(* Schneider Machine Expert - Basic project Modelo final v1.2, file version 2.5.0.0 *)
(* ProjectInformations: Name=Nuevo proyecto *)

HARDWARE
  Cpu 0: TM221CE24T
  EthernetConfiguration: NetworkName=M221, IpAllocationMode=FixedAddress, IpAddress=0.0.0.0, SubnetMask=0.0.0.0
  SerialLineConfiguration: Baud=Baud19200, Parity=ParityEven, DataBits=DataBits8, StopBits=StopBits1, PhysicalMedium=PhysicalMediumRs485, TransmissionMode=TransmissionModeModbusRtu, SlaveId=1, Addressing=SlaveAddressing
  MastTask: UsePeriodScanMode=false, PeriodScan=100
  FastTask: Period=255
  CpuBehavior: StartingMode=StartAsPreviousState, AutoSaveRamOnEeprom=true, WatchdogPeriod=250

SYMBOLS  (address, symbol, comment, settings)
  %M0         "Escalon frontal izquierdo"
  %M1         "Escalon frontal derecho"
  %M2         "Escalon trasero izquierdo"
  %M3         "Escalon trasero derecho"
  %M4         "Sensor frente izquierdo"
  %M5         "Sensor frente medio"
  %M6         "Sensor frente derecho"
  %M7         "Sensor derecha adelante"
  %M8         "Sensor derecha medio"
  %M9         "Sensor derecha atras"
  %M10        "Sensor trasero derecha"
  %M11        "Sensor trasero medio"
  %M12        "Sensor trasero izquierda"
  %M13        "Sensor izquierda atras"
  %M14        "Sensor izquierda medio"
  %M15        "Sensor izquierda adelante"
  %M16      FIFO_IN  "Carga en fifo"
  %M17      FIFO_OUT  "Descarga de fifo"
  %M40      RST_S  "Reset/Enable Generador S"
  %M41      RST_DEMUX  "Reset/Enbale Demux"
  %M42      EN_ENCOD  "Enable Encoders"
  %M43      RST_ENCOD  "Reset Encoders"
  %M44      RST_FIFO  "Reset FIFOS"
  %M45      RST_STOP
  %M50      STP_MOV  "Stop Movement"
  %M51        "Enable Forward"
  %M52        "Enable Giro Horario"
  %M53        "Enable Giro A-Horario"
  %M54        "Enable F-G-H"
  %M55        "Enable F-G-AH"
  %M56        "Enable B-G-H"
  %M57        "Enable B-G-AH"
  %S6       SB_TB1S  "Base de tiempo de 1 s generada por un reloj interno"
  %MW10       "Comando Rueda Izquierda"
  %MW11       "Comando Rueda Derecha"
  %MW12       "Velocidad Rueda Izquierda"
  %MW13       "Velocidad Rueda Derecha"
  %TM0        [Preset=5, Base=OneHundredMilliSeconds]
  %TM1        [Preset=5, Base=OneHundredMilliSeconds]
  %TM2        [Preset=5, Base=OneHundredMilliSeconds]
  %TM3        [Preset=5, Base=OneHundredMilliSeconds]
  %TM4        [Preset=5, Base=OneHundredMilliSeconds]
  %TM5        [Preset=5, Base=OneHundredMilliSeconds]
  %TM6        [Preset=5, Base=OneHundredMilliSeconds]
  %TM7        [Preset=5, Base=OneHundredMilliSeconds]
  %TM8        [Preset=5, Base=OneHundredMilliSeconds]
  %TM9        [Preset=5, Base=OneHundredMilliSeconds]
  %TM10       [Preset=5, Base=OneHundredMilliSeconds]
  %TM11       [Preset=5, Base=OneHundredMilliSeconds]
  %TM12       [Preset=5, Base=OneHundredMilliSeconds]
  %TM13       [Preset=5, Base=OneHundredMilliSeconds]
  %TM14       [Preset=5, Base=OneHundredMilliSeconds]
  %TM15       [Preset=5, Base=OneHundredMilliSeconds]
  %C0         [Preset=17]
  %R0         "Pasos Izquierda"
  %R1         "Pasos Derecha"
  %R2         "Velocidad Izquierda"
  %R3         "Velocidad Derecha"
  %UDF0.RETF0   "Orientacion"  [CompiledType=Float, Type=ReturnValue, DisplayedAddress=%RET0, CompiledAddress=%UDFRETURNF0]
  %UDF0.VARF0   "Cuenta encoder L"  [CompiledType=Float, Type=Variable, DisplayedAddress=%VAR0, CompiledAddress=%UDFVARF0]
  %UDF0.VARF1   "Cuenta Encoder R"  [CompiledType=Float, Type=Variable, DisplayedAddress=%VAR1, CompiledAddress=%UDFVARF1]
  %UDF0.VARF2   "Radio de la Rueda"  [CompiledType=Float, Type=Variable, DisplayedAddress=%VAR2, CompiledAddress=%UDFVARF2]
  %UDF0.VARF4   "Pasos"  [CompiledType=Float, Type=Variable, DisplayedAddress=%VAR4, CompiledAddress=%UDFVARF4]
  %UDF0.VARF6   "ΔSL"  [CompiledType=Float, Type=Variable, DisplayedAddress=%VAR6, CompiledAddress=%UDFVARF6]
  %UDF0.VARF7   "ΔSR:"  [CompiledType=Float, Type=Variable, DisplayedAddress=%VAR7, CompiledAddress=%UDFVARF7]
  %UDF0.VARF9   "Longitud Eje"  [CompiledType=Float, Type=Variable, DisplayedAddress=%VAR9, CompiledAddress=%UDFVARF9]
  %I0.0     ENC1A  "Input"
  %I0.1     ENC1B  "Enable"
  %I0.6     ENC2A
  %I0.7     ENC2B
  %I0.8     MUX_IN  "Data de mux sensores"
  %Q0.0     L_PWM  "Salida PWM Motor Izquierdo"
  %Q0.1     R_PWM  "Salida PWM Motor Derecho"
  %Q0.2     L_DIR  "Salida Direccion Motor Izquierdo - 0:F 1:B"
  %Q0.3     R_DIR  "Salida Direccion Motor Derecho - 0:F 1:B"
  %Q0.4     S0  "MUX S0"
  %Q0.5     S1  "MUX S1"
  %Q0.6     S2  "MUX S2"
  %Q0.7     S3  "MUX S3"
  %Q0.8       "LAMPARAS BIT 0"
  %Q0.9       "LAMPARAS BIT 1"
  %HSC0       "Encoder Rueda Izquierda"  [Type=CounterOrDownCounterBiPhasesX2, Preset=0, UseDoubleWord=true, DedicatedInputs(DedicatedInput(Activated=true), DedicatedInput(Activated=true)), ReflexOutputs(ReflexOutput(Activated=false, LessThanS0=false, GreaterOrEqualThanS0=false, GreaterOrEqualThanS1=false), ReflexOutput(Activated=false, LessThanS0=false, GreaterOrEqualThanS0=false, GreaterOrEqualThanS1=false)), Thresholds(Threshold(Thresh]
  %HSC1       "Encoder Rueda Derecha"  [Type=CounterOrDownCounterBiPhasesX2, Preset=0, UseDoubleWord=true, DedicatedInputs(DedicatedInput(Activated=true), DedicatedInput(Activated=true)), ReflexOutputs(ReflexOutput(Activated=false, LessThanS0=false, GreaterOrEqualThanS0=false, GreaterOrEqualThanS1=false), ReflexOutput(Activated=false, LessThanS0=false, GreaterOrEqualThanS0=false, GreaterOrEqualThanS1=false)), Thresholds(Threshold(Thresh]
  %PWM0       "PWM_L"  [PtoObject(RefInput=NotUsed, ZPhaseInput=NotUsed, ProbeInput=NotUsed), GlobalIndex=0, Type=PWM, TimeBase=OneMilliSeconds, Preset=1]
  %PWM1       "PWM_R"  [PtoObject(RefInput=NotUsed, ZPhaseInput=NotUsed, ProbeInput=NotUsed), GlobalIndex=1, Type=PWM, TimeBase=OneMilliSeconds, Preset=1]

POU Demux
  (* SectionNumber=1 *)

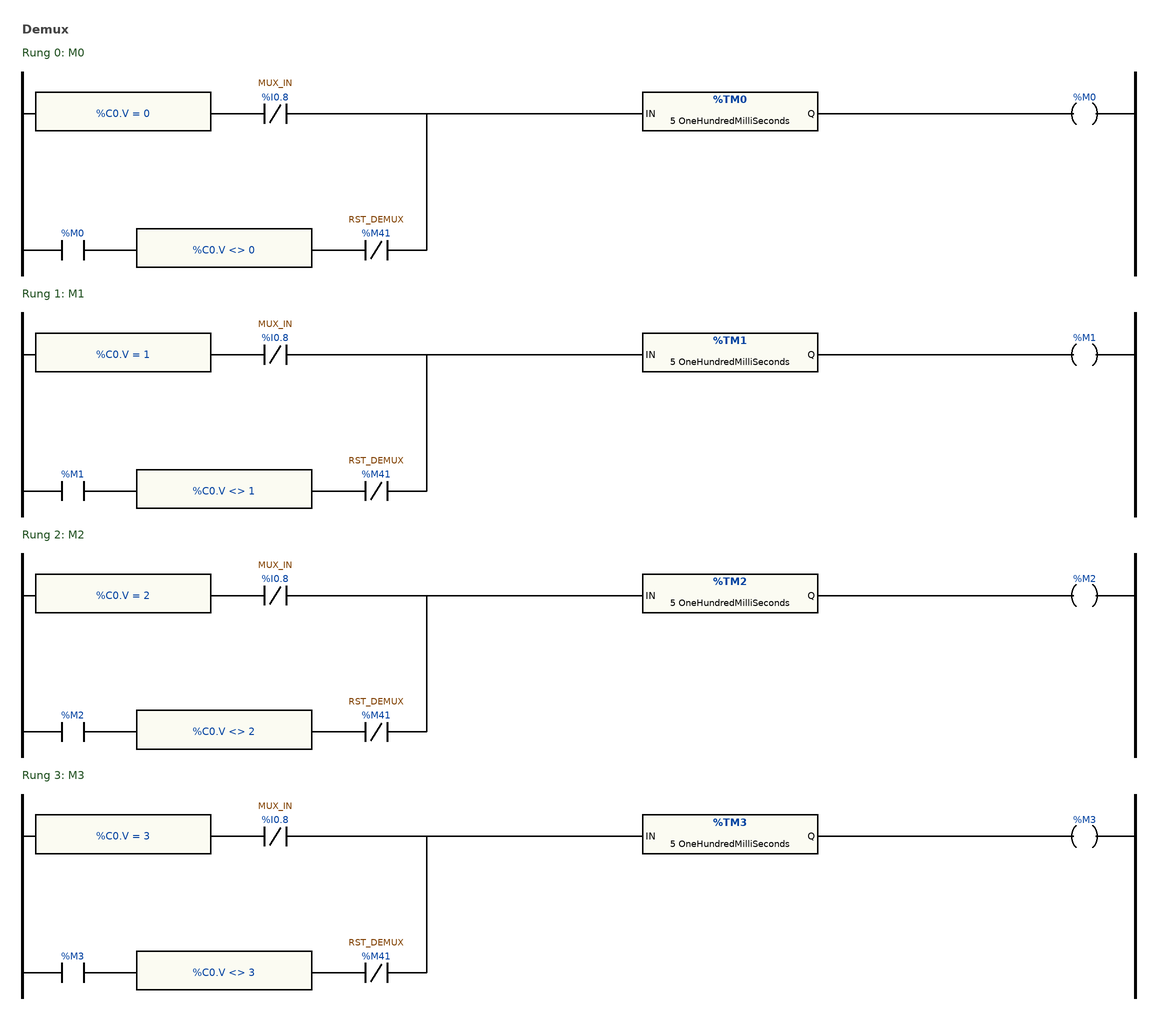

// Rung 0: M0
  BLK %TM0
  LD [ %C0.V = 0 ]
  ANDN %I0.8              (* MUX_IN *)
  OR( %M0
  AND [ %C0.V <> 0 ]
  ANDN %M41               (* RST_DEMUX *)
  )
  IN
  OUT_BLK
  LD Q
  ST %M0
  END_BLK
  // as ST:
  //   %TM0(IN := %C0.V = 0 AND NOT MUX_IN OR %M0 AND %C0.V <> 0 AND NOT RST_DEMUX);
  //   %M0 := %TM0.Q;

// Rung 1: M1
  BLK %TM1
  LD [ %C0.V = 1 ]
  ANDN %I0.8              (* MUX_IN *)
  OR( %M1
  AND [ %C0.V <> 1 ]
  ANDN %M41               (* RST_DEMUX *)
  )
  IN
  OUT_BLK
  LD Q
  ST %M1
  END_BLK
  // as ST:
  //   %TM1(IN := %C0.V = 1 AND NOT MUX_IN OR %M1 AND %C0.V <> 1 AND NOT RST_DEMUX);
  //   %M1 := %TM1.Q;

// Rung 2: M2
  BLK %TM2
  LD [ %C0.V = 2 ]
  ANDN %I0.8              (* MUX_IN *)
  OR( %M2
  AND [ %C0.V <> 2 ]
  ANDN %M41               (* RST_DEMUX *)
  )
  IN
  OUT_BLK
  LD Q
  ST %M2
  END_BLK
  // as ST:
  //   %TM2(IN := %C0.V = 2 AND NOT MUX_IN OR %M2 AND %C0.V <> 2 AND NOT RST_DEMUX);
  //   %M2 := %TM2.Q;

// Rung 3: M3
  BLK %TM3
  LD [ %C0.V = 3 ]
  ANDN %I0.8              (* MUX_IN *)
  OR( %M3
  AND [ %C0.V <> 3 ]
  ANDN %M41               (* RST_DEMUX *)
  )
  IN
  OUT_BLK
  LD Q
  ST %M3
  END_BLK
  // as ST:
  //   %TM3(IN := %C0.V = 3 AND NOT MUX_IN OR %M3 AND %C0.V <> 3 AND NOT RST_DEMUX);
  //   %M3 := %TM3.Q;

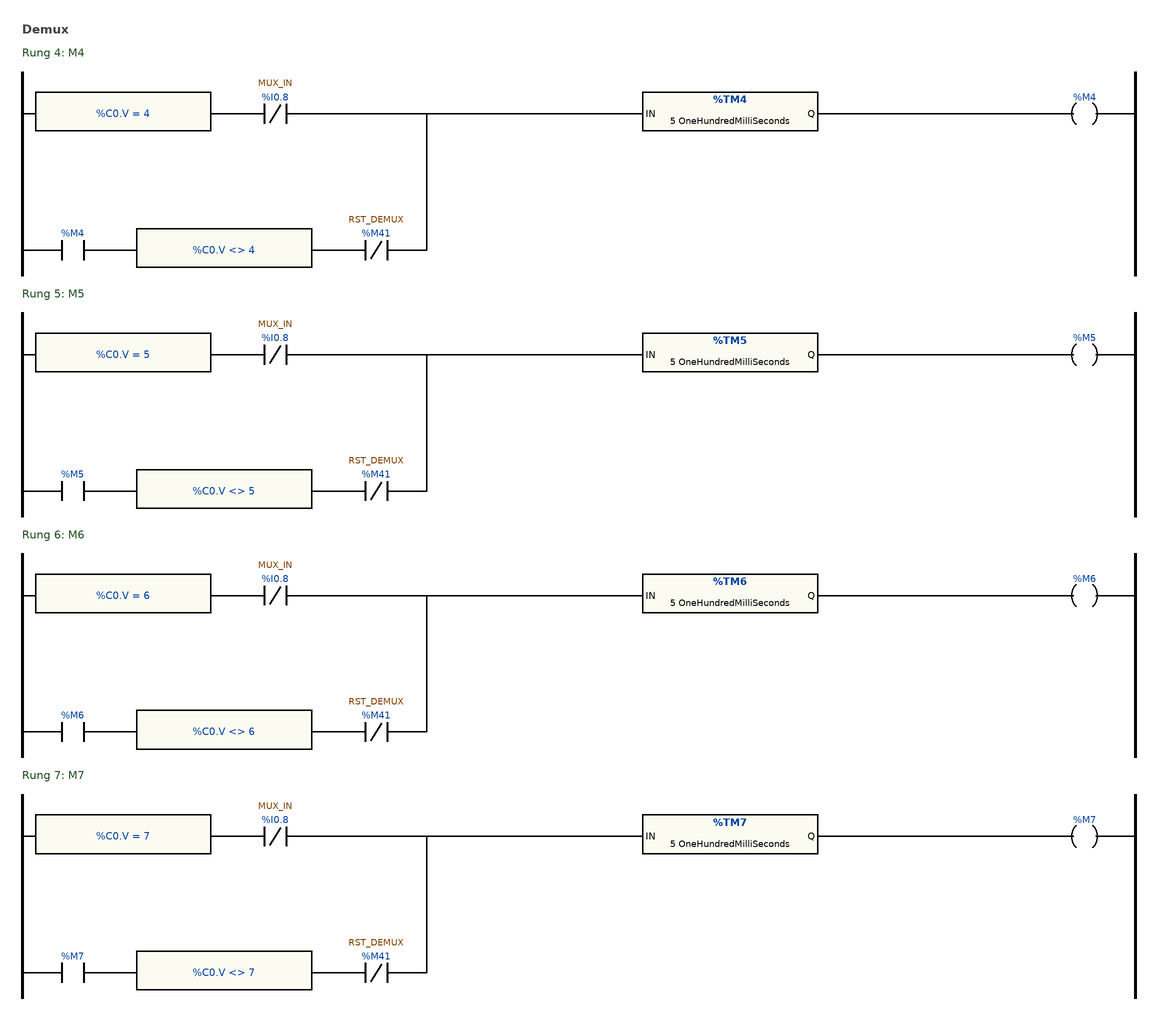

// Rung 4: M4
  BLK %TM4
  LD [ %C0.V = 4 ]
  ANDN %I0.8              (* MUX_IN *)
  OR( %M4
  AND [ %C0.V <> 4 ]
  ANDN %M41               (* RST_DEMUX *)
  )
  IN
  OUT_BLK
  LD Q
  ST %M4
  END_BLK
  // as ST:
  //   %TM4(IN := %C0.V = 4 AND NOT MUX_IN OR %M4 AND %C0.V <> 4 AND NOT RST_DEMUX);
  //   %M4 := %TM4.Q;

// Rung 5: M5
  BLK %TM5
  LD [ %C0.V = 5 ]
  ANDN %I0.8              (* MUX_IN *)
  OR( %M5
  AND [ %C0.V <> 5 ]
  ANDN %M41               (* RST_DEMUX *)
  )
  IN
  OUT_BLK
  LD Q
  ST %M5
  END_BLK
  // as ST:
  //   %TM5(IN := %C0.V = 5 AND NOT MUX_IN OR %M5 AND %C0.V <> 5 AND NOT RST_DEMUX);
  //   %M5 := %TM5.Q;

// Rung 6: M6
  BLK %TM6
  LD [ %C0.V = 6 ]
  ANDN %I0.8              (* MUX_IN *)
  OR( %M6
  AND [ %C0.V <> 6 ]
  ANDN %M41               (* RST_DEMUX *)
  )
  IN
  OUT_BLK
  LD Q
  ST %M6
  END_BLK
  // as ST:
  //   %TM6(IN := %C0.V = 6 AND NOT MUX_IN OR %M6 AND %C0.V <> 6 AND NOT RST_DEMUX);
  //   %M6 := %TM6.Q;

// Rung 7: M7
  BLK %TM7
  LD [ %C0.V = 7 ]
  ANDN %I0.8              (* MUX_IN *)
  OR( %M7
  AND [ %C0.V <> 7 ]
  ANDN %M41               (* RST_DEMUX *)
  )
  IN
  OUT_BLK
  LD Q
  ST %M7
  END_BLK
  // as ST:
  //   %TM7(IN := %C0.V = 7 AND NOT MUX_IN OR %M7 AND %C0.V <> 7 AND NOT RST_DEMUX);
  //   %M7 := %TM7.Q;

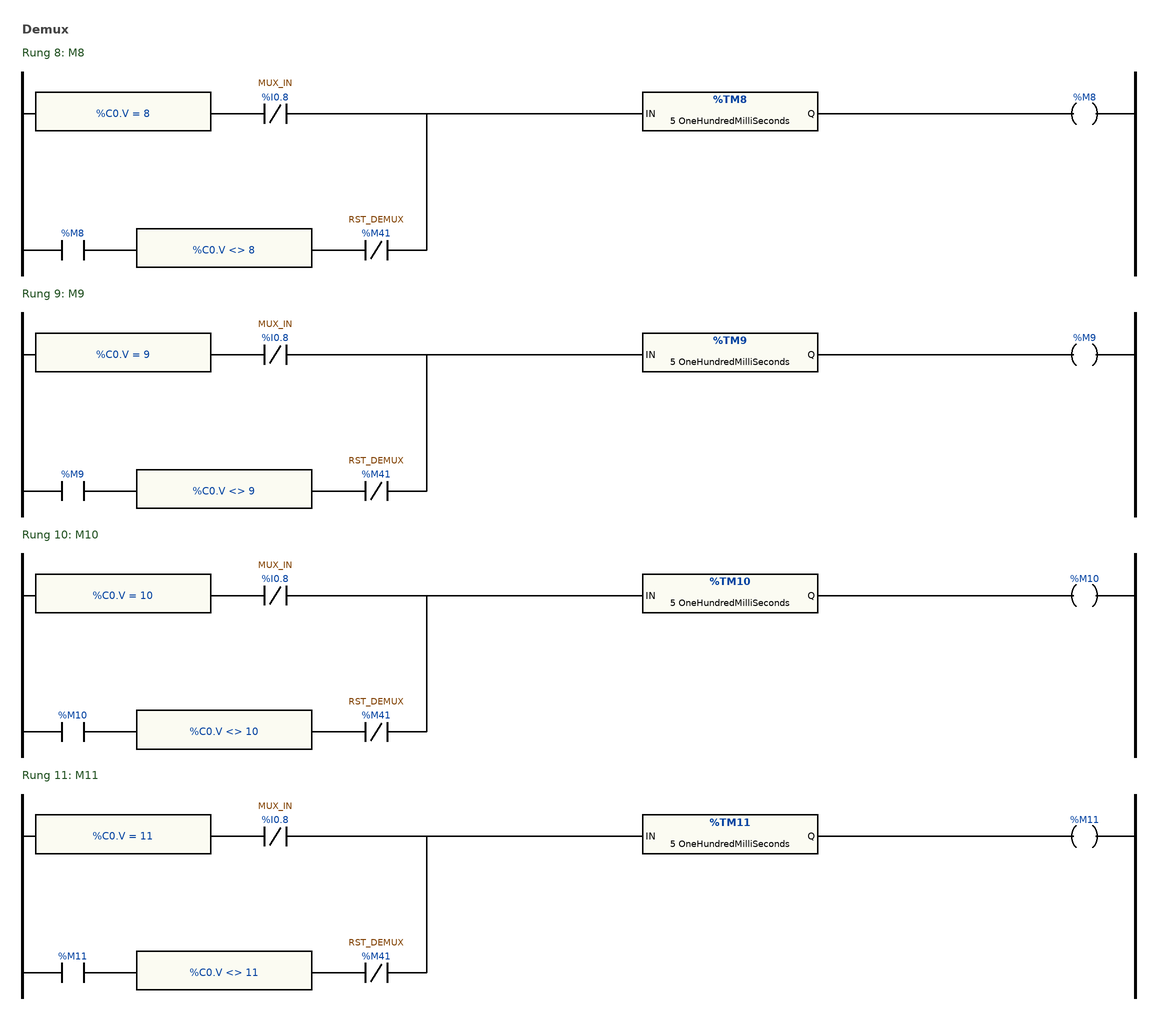

// Rung 8: M8
  BLK %TM8
  LD [ %C0.V = 8 ]
  ANDN %I0.8              (* MUX_IN *)
  OR( %M8
  AND [ %C0.V <> 8 ]
  ANDN %M41               (* RST_DEMUX *)
  )
  IN
  OUT_BLK
  LD Q
  ST %M8
  END_BLK
  // as ST:
  //   %TM8(IN := %C0.V = 8 AND NOT MUX_IN OR %M8 AND %C0.V <> 8 AND NOT RST_DEMUX);
  //   %M8 := %TM8.Q;

// Rung 9: M9
  BLK %TM9
  LD [ %C0.V = 9 ]
  ANDN %I0.8              (* MUX_IN *)
  OR( %M9
  AND [ %C0.V <> 9 ]
  ANDN %M41               (* RST_DEMUX *)
  )
  IN
  OUT_BLK
  LD Q
  ST %M9
  END_BLK
  // as ST:
  //   %TM9(IN := %C0.V = 9 AND NOT MUX_IN OR %M9 AND %C0.V <> 9 AND NOT RST_DEMUX);
  //   %M9 := %TM9.Q;

// Rung 10: M10
  BLK %TM10
  LD [ %C0.V = 10 ]
  ANDN %I0.8              (* MUX_IN *)
  OR( %M10
  AND [ %C0.V <> 10 ]
  ANDN %M41               (* RST_DEMUX *)
  )
  IN
  OUT_BLK
  LD Q
  ST %M10
  END_BLK
  // as ST:
  //   %TM10(IN := %C0.V = 10 AND NOT MUX_IN OR %M10 AND %C0.V <> 10 AND NOT RST_DEMUX);
  //   %M10 := %TM10.Q;

// Rung 11: M11
  BLK %TM11
  LD [ %C0.V = 11 ]
  ANDN %I0.8              (* MUX_IN *)
  OR( %M11
  AND [ %C0.V <> 11 ]
  ANDN %M41               (* RST_DEMUX *)
  )
  IN
  OUT_BLK
  LD Q
  ST %M11
  END_BLK
  // as ST:
  //   %TM11(IN := %C0.V = 11 AND NOT MUX_IN OR %M11 AND %C0.V <> 11 AND NOT RST_DEMUX);
  //   %M11 := %TM11.Q;

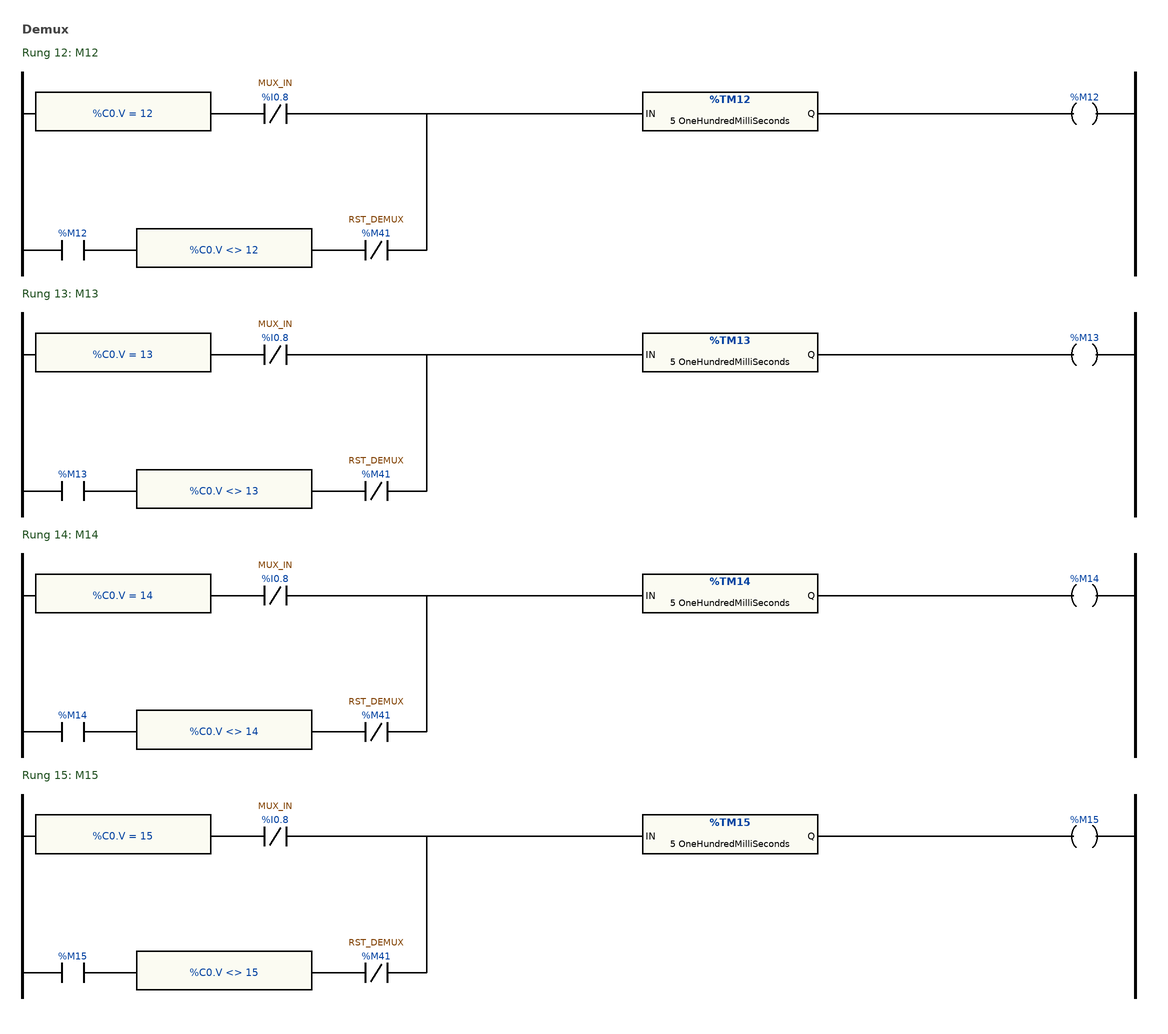

// Rung 12: M12
  BLK %TM12
  LD [ %C0.V = 12 ]
  ANDN %I0.8              (* MUX_IN *)
  OR( %M12
  AND [ %C0.V <> 12 ]
  ANDN %M41               (* RST_DEMUX *)
  )
  IN
  OUT_BLK
  LD Q
  ST %M12
  END_BLK
  // as ST:
  //   %TM12(IN := %C0.V = 12 AND NOT MUX_IN OR %M12 AND %C0.V <> 12 AND NOT RST_DEMUX);
  //   %M12 := %TM12.Q;

// Rung 13: M13
  BLK %TM13
  LD [ %C0.V = 13 ]
  ANDN %I0.8              (* MUX_IN *)
  OR( %M13
  AND [ %C0.V <> 13 ]
  ANDN %M41               (* RST_DEMUX *)
  )
  IN
  OUT_BLK
  LD Q
  ST %M13
  END_BLK
  // as ST:
  //   %TM13(IN := %C0.V = 13 AND NOT MUX_IN OR %M13 AND %C0.V <> 13 AND NOT RST_DEMUX);
  //   %M13 := %TM13.Q;

// Rung 14: M14
  BLK %TM14
  LD [ %C0.V = 14 ]
  ANDN %I0.8              (* MUX_IN *)
  OR( %M14
  AND [ %C0.V <> 14 ]
  ANDN %M41               (* RST_DEMUX *)
  )
  IN
  OUT_BLK
  LD Q
  ST %M14
  END_BLK
  // as ST:
  //   %TM14(IN := %C0.V = 14 AND NOT MUX_IN OR %M14 AND %C0.V <> 14 AND NOT RST_DEMUX);
  //   %M14 := %TM14.Q;

// Rung 15: M15
  BLK %TM15
  LD [ %C0.V = 15 ]
  ANDN %I0.8              (* MUX_IN *)
  OR( %M15
  AND [ %C0.V <> 15 ]
  ANDN %M41               (* RST_DEMUX *)
  )
  IN
  OUT_BLK
  LD Q
  ST %M15
  END_BLK
  // as ST:
  //   %TM15(IN := %C0.V = 15 AND NOT MUX_IN OR %M15 AND %C0.V <> 15 AND NOT RST_DEMUX);
  //   %M15 := %TM15.Q;

POU Generacion Sx
  (* SectionNumber=2 *)

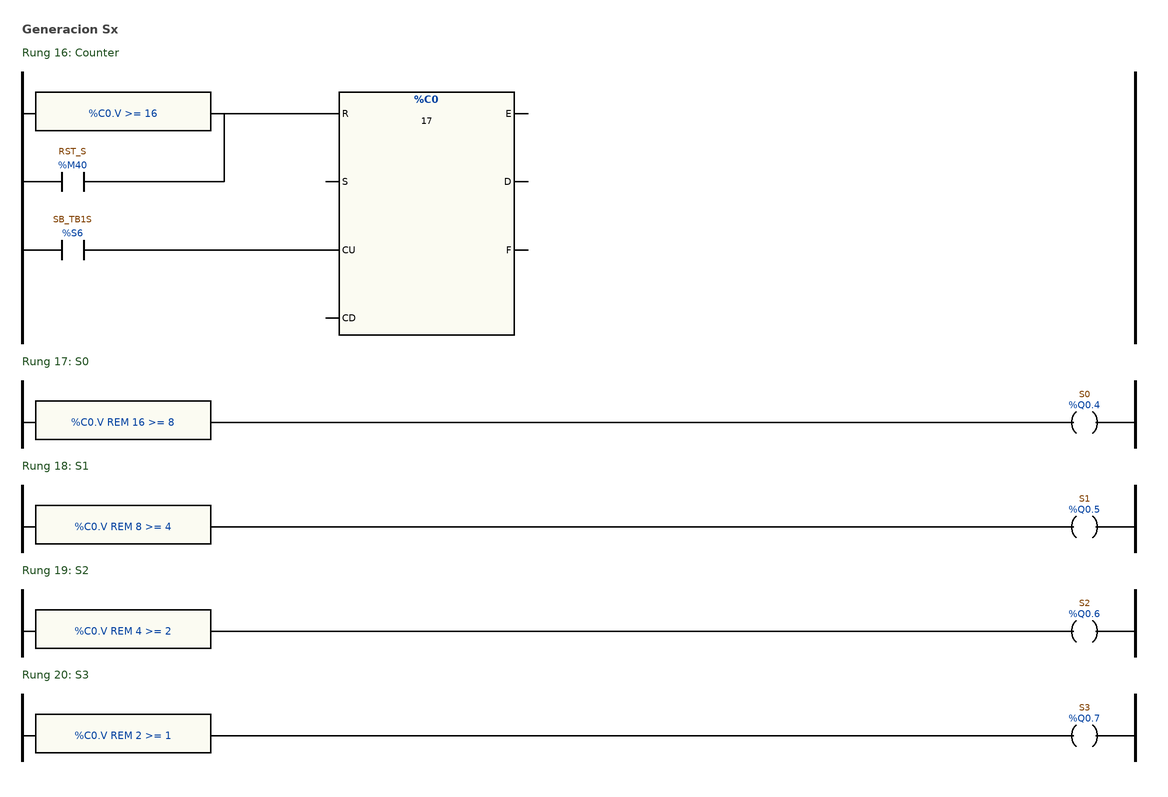

// Rung 16: Counter
  BLK %C0
  LD [ %C0.V >= 16 ]
  OR %M40                 (* RST_S *)
  R
  LD %S6                  (* SB_TB1S *)
  CU
  END_BLK
  // as ST:
  //   %C0(R := %C0.V >= 16 OR RST_S, CU := SB_TB1S);

// Rung 17: S0
  LD 1
  AND [%C0.V REM 16 >= 8]
  ST %Q0.4                (* S0 *)
  // as ST:
  //   S0 := %C0.V REM 16 >= 8;

// Rung 18: S1
  LD 1
  AND [%C0.V REM 8 >= 4]
  ST %Q0.5                (* S1 *)
  // as ST:
  //   S1 := %C0.V REM 8 >= 4;

// Rung 19: S2
  LD 1
  AND [%C0.V REM 4 >= 2]
  ST %Q0.6                (* S2 *)
  // as ST:
  //   S2 := %C0.V REM 4 >= 2;

// Rung 20: S3
  LD 1
  AND [%C0.V REM 2 >= 1]
  ST %Q0.7                (* S3 *)
  // as ST:
  //   S3 := %C0.V REM 2 >= 1;

POU Encoders
  (* SectionNumber=0 *)

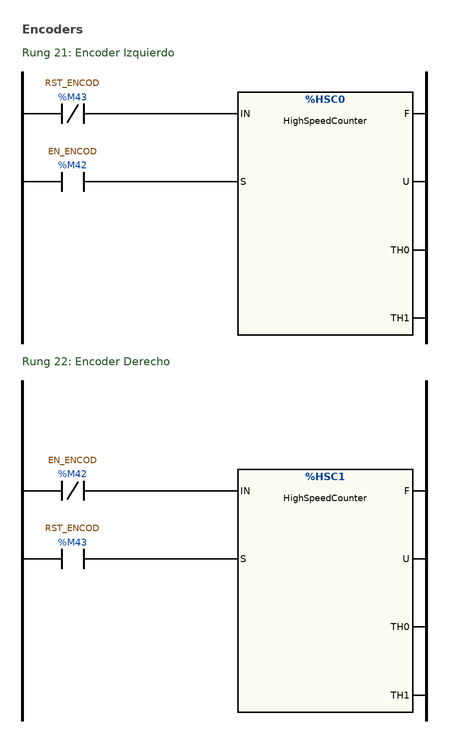

// Rung 21: Encoder Izquierdo
  BLK %HSC0
  LDN %M43                (* RST_ENCOD *)
  IN
  LD %M42                 (* EN_ENCOD *)
  S
  END_BLK
  // as ST:
  //   %HSC0(IN := NOT RST_ENCOD, S := EN_ENCOD);

// Rung 22: Encoder Derecho
  BLK %HSC1
  LDN %M42                (* EN_ENCOD *)
  IN
  LD %M43                 (* RST_ENCOD *)
  S
  END_BLK
  // as ST:
  //   %HSC1(IN := NOT EN_ENCOD, S := RST_ENCOD);

POU Control de Motores
  (* SectionNumber=0 *)

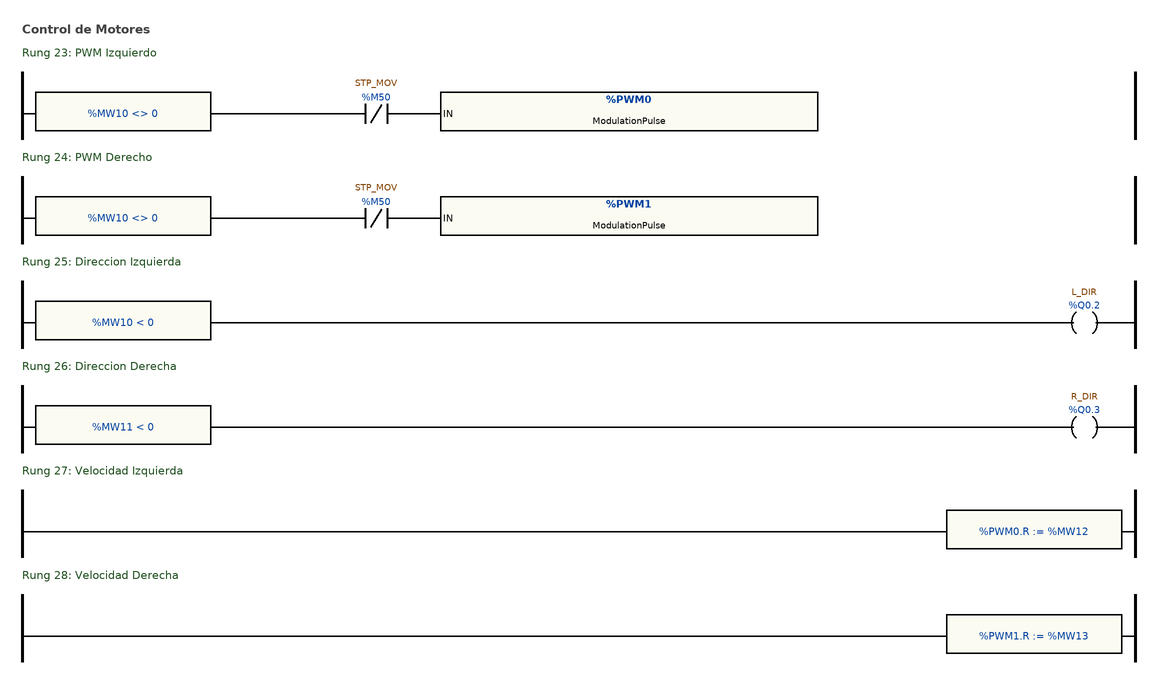

// Rung 23: PWM Izquierdo
  BLK %PWM0
  LD [ %MW10 <> 0 ]
  ANDN %M50               (* STP_MOV *)
  IN
  END_BLK
  // as ST:
  //   %PWM0(IN := %MW10 <> 0 AND NOT STP_MOV);

// Rung 24: PWM Derecho
  BLK %PWM1
  LD [ %MW10 <> 0 ]
  ANDN %M50               (* STP_MOV *)
  IN
  END_BLK
  // as ST:
  //   %PWM1(IN := %MW10 <> 0 AND NOT STP_MOV);

// Rung 25: Direccion Izquierda
  LD [ %MW10 < 0 ]
  ST %Q0.2                (* L_DIR *)
  // as ST:
  //   L_DIR := %MW10 < 0;

// Rung 26: Direccion Derecha
  LD [ %MW11 < 0 ]
  ST %Q0.3                (* R_DIR *)
  // as ST:
  //   R_DIR := %MW11 < 0;

// Rung 27: Velocidad Izquierda
  LD 1
  [ %PWM0.R := %MW12 ]
  // as ST:
  //   %PWM0.R := %MW12;

// Rung 28: Velocidad Derecha
  LD 1
  [ %PWM1.R := %MW13 ]
  // as ST:
  //   %PWM1.R := %MW13;

POU FIFOS
  (* SectionNumber=0 *)

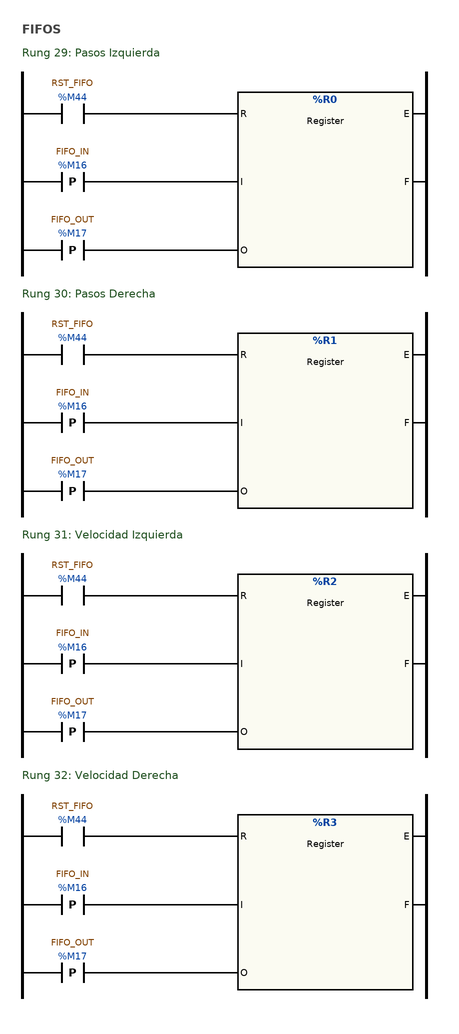

// Rung 29: Pasos Izquierda
  BLK %R0
  LD %M44                 (* RST_FIFO *)
  R
  LDR %M16                (* FIFO_IN *)
  I
  LDR %M17                (* FIFO_OUT *)
  O
  END_BLK
  // as ST:
  //   %R0(R := RST_FIFO, I := RISING(FIFO_IN), O := RISING(FIFO_OUT));

// Rung 30: Pasos Derecha
  BLK %R1
  LD %M44                 (* RST_FIFO *)
  R
  LDR %M16                (* FIFO_IN *)
  I
  LDR %M17                (* FIFO_OUT *)
  O
  END_BLK
  // as ST:
  //   %R1(R := RST_FIFO, I := RISING(FIFO_IN), O := RISING(FIFO_OUT));

// Rung 31: Velocidad Izquierda
  BLK %R2
  LD %M44                 (* RST_FIFO *)
  R
  LDR %M16                (* FIFO_IN *)
  I
  LDR %M17                (* FIFO_OUT *)
  O
  END_BLK
  // as ST:
  //   %R2(R := RST_FIFO, I := RISING(FIFO_IN), O := RISING(FIFO_OUT));

// Rung 32: Velocidad Derecha
  BLK %R3
  LD %M44                 (* RST_FIFO *)
  R
  LDR %M16                (* FIFO_IN *)
  I
  LDR %M17                (* FIFO_OUT *)
  O
  END_BLK
  // as ST:
  //   %R3(R := RST_FIFO, I := RISING(FIFO_IN), O := RISING(FIFO_OUT));

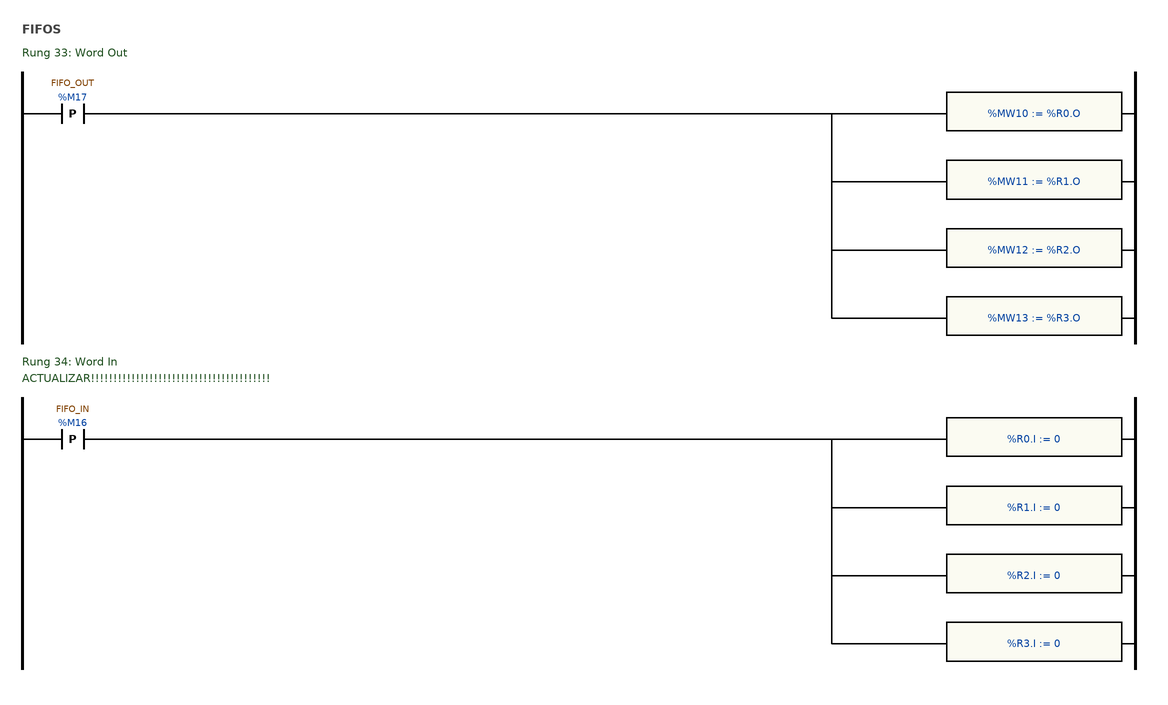

// Rung 33: Word Out
  LDR %M17                (* FIFO_OUT *)
  [ %MW10 := %R0.O ]
  [ %MW11 := %R1.O ]
  [ %MW12 := %R2.O ]
  [ %MW13 := %R3.O ]
  // as ST:
  //   IF RISING(FIFO_OUT) THEN %MW10 := %R0.O; END_IF;
  //   IF RISING(FIFO_OUT) THEN %MW11 := %R1.O; END_IF;
  //   IF RISING(FIFO_OUT) THEN %MW12 := %R2.O; END_IF;
  //   IF RISING(FIFO_OUT) THEN %MW13 := %R3.O; END_IF;

// Rung 34: Word In
// ACTUALIZAR!!!!!!!!!!!!!!!!!!!!!!!!!!!!!!!!!!!!!!!!
  LDR %M16                (* FIFO_IN *)
  [ %R0.I := 0 ]
  [ %R1.I := 0 ]
  [ %R2.I := 0 ]
  [ %R3.I := 0 ]
  // as ST:
  //   IF RISING(FIFO_IN) THEN %R0.I := 0; END_IF;
  //   IF RISING(FIFO_IN) THEN %R1.I := 0; END_IF;
  //   IF RISING(FIFO_IN) THEN %R2.I := 0; END_IF;
  //   IF RISING(FIFO_IN) THEN %R3.I := 0; END_IF;

POU Control de Colision
  (* SectionNumber=0 *)

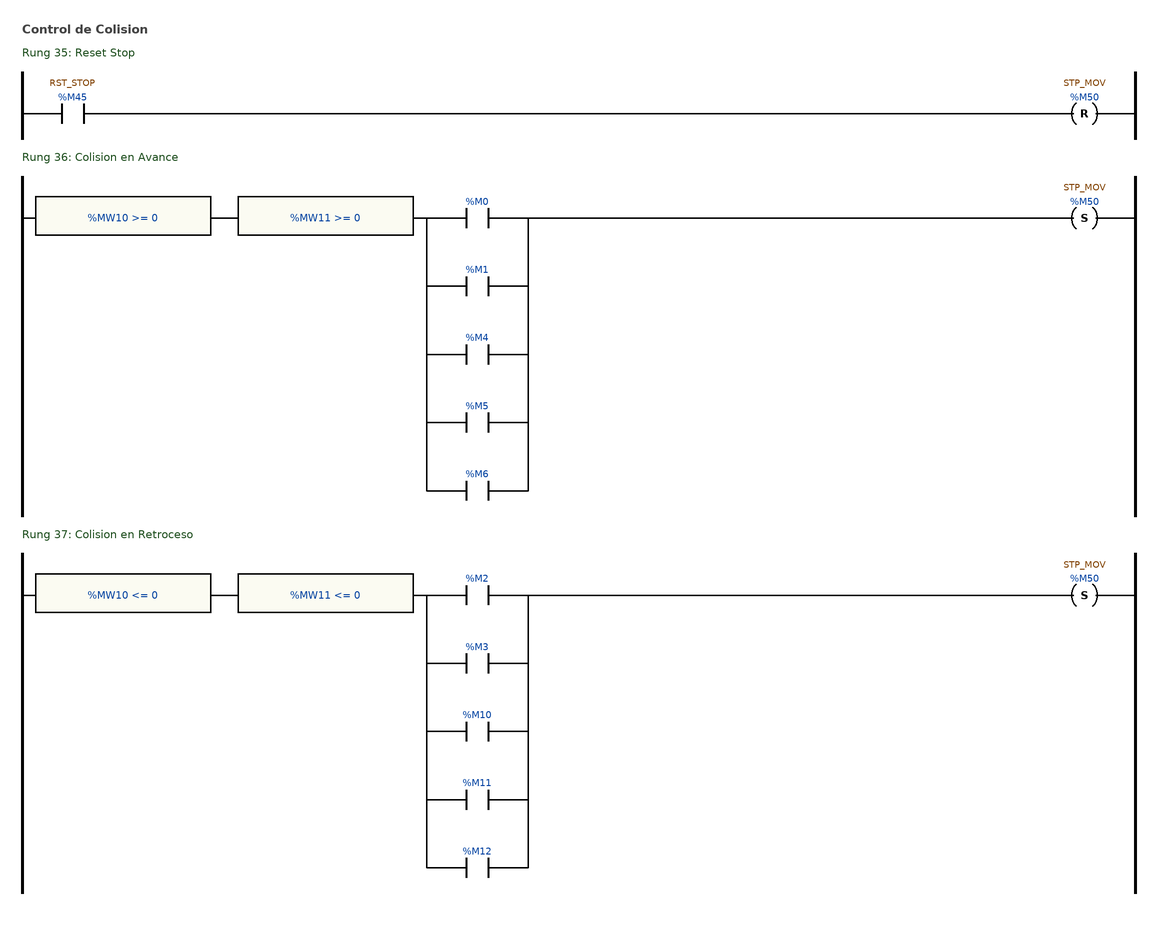

// Rung 35: Reset Stop
  LD %M45                 (* RST_STOP *)
  R %M50                  (* STP_MOV *)
  // as ST:
  //   IF RST_STOP THEN STP_MOV := FALSE; END_IF;

// Rung 36: Colision en Avance
  LD [ %MW10 >= 0 ]
  AND [ %MW11 >= 0 ]
  AND( %M0
  OR %M1
  OR %M4
  OR %M5
  OR %M6
  )
  S %M50                  (* STP_MOV *)
  // as ST:
  //   IF %MW10 >= 0 AND %MW11 >= 0 AND (%M0 OR %M1 OR %M4 OR %M5 OR %M6) THEN STP_MOV := TRUE; END_IF;

// Rung 37: Colision en Retroceso
  LD [ %MW10 <= 0 ]
  AND [ %MW11 <= 0 ]
  AND( %M2
  OR %M3
  OR %M10
  OR %M11
  OR %M12
  )
  S %M50                  (* STP_MOV *)
  // as ST:
  //   IF %MW10 <= 0 AND %MW11 <= 0 AND (%M2 OR %M3 OR %M10 OR %M11 OR %M12) THEN STP_MOV := TRUE; END_IF;

UserFunctionPou ORIENTACION
  (* SectionNumber=2, Description=%RET0: Orientacion
%PARAM0: Cuenta encoder L
%PARAM1: Cuenta encoder R
ΔSL: Avanze lineal Rueda Izquierda
ΔSR: Avanze lineal Rueda Derecha *)

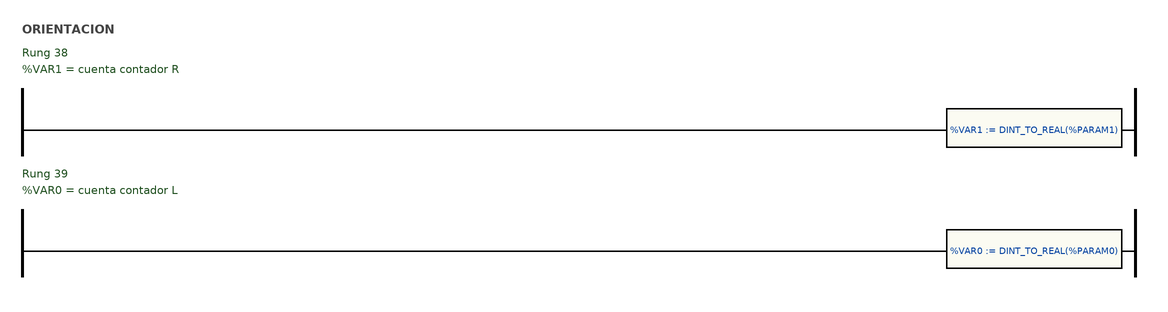

// Rung 38
// %VAR1 = cuenta contador R
  LD 1
  [%VAR1 := DINT_TO_REAL(%PARAM1)]
  // as ST:
  //   %VAR1 := DINT_TO_REAL(%PARAM1);

// Rung 39
// %VAR0 = cuenta contador L
  LD 1
  [%VAR0 := DINT_TO_REAL(%PARAM0)]
  // as ST:
  //   %VAR0 := DINT_TO_REAL(%PARAM0);

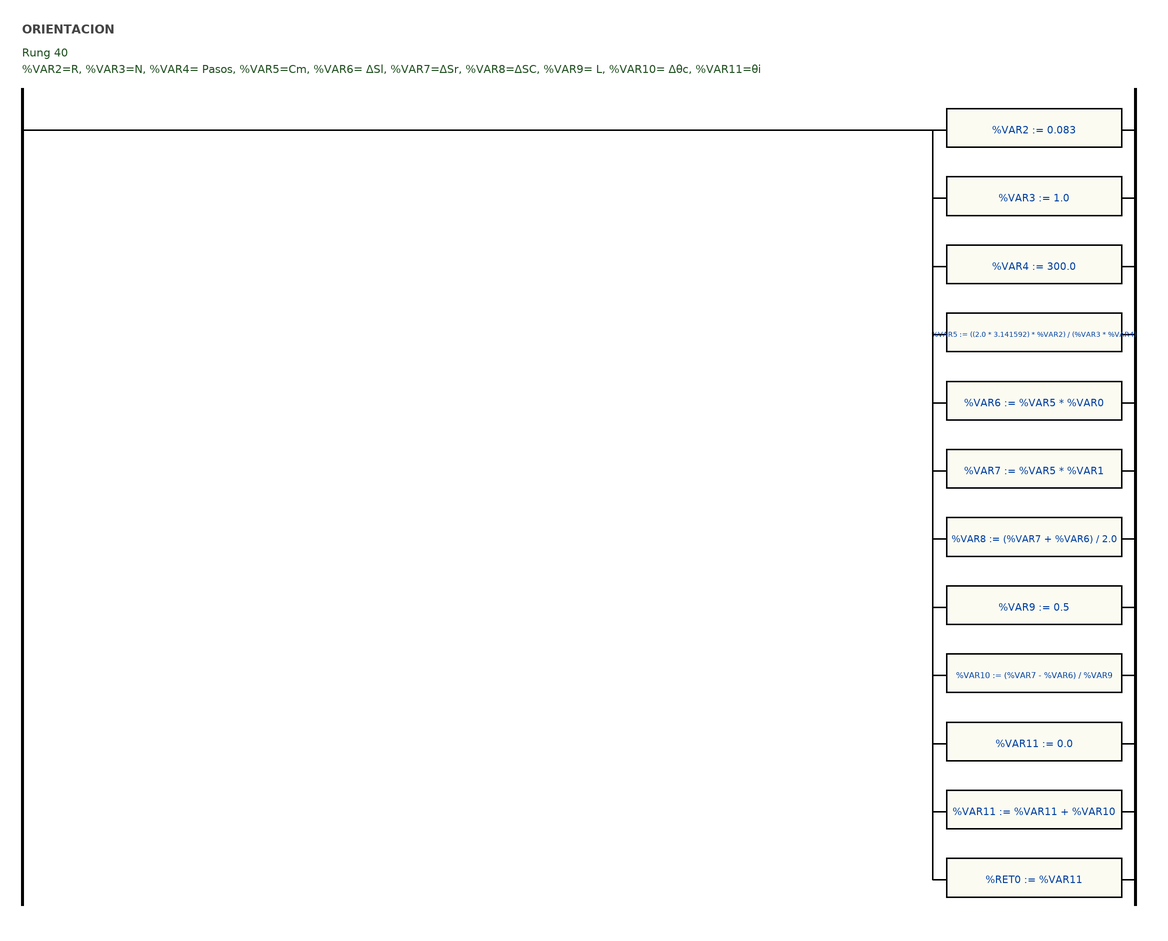

// Rung 40
// %VAR2=R, %VAR3=N, %VAR4= Pasos, %VAR5=Cm, %VAR6= ΔSl, %VAR7=ΔSr, %VAR8=ΔSC, %VAR9= L, %VAR10= Δθc, %VAR11=θi
  LD 1
  [%VAR2 := 0.083]
  [%VAR3 := 1.0]
  [%VAR4 := 300.0]
  [%VAR5 := ((2.0 * 3.141592) * %VAR2) / (%VAR3 * %VAR4)]
  [%VAR6 := %VAR5 * %VAR0]
  [%VAR7 := %VAR5 * %VAR1]
  [%VAR8 := (%VAR7 + %VAR6) / 2.0]
  [%VAR9 := 0.5]
  [%VAR10 := (%VAR7 - %VAR6) / %VAR9]
  [%VAR11 := 0.0]
  [%VAR11 := %VAR11 + %VAR10]
  [%RET0 := %VAR11]
  // as ST:
  //   %VAR2 := 0.083;
  //   %VAR3 := 1.0;
  //   %VAR4 := 300.0;
  //   %VAR5 := ((2.0 * 3.141592) * %VAR2) / (%VAR3 * %VAR4);
  //   %VAR6 := %VAR5 * %VAR0;
  //   %VAR7 := %VAR5 * %VAR1;
  //   %VAR8 := (%VAR7 + %VAR6) / 2.0;
  //   %VAR9 := 0.5;
  //   %VAR10 := (%VAR7 - %VAR6) / %VAR9;
  //   %VAR11 := 0.0;
  //   %VAR11 := %VAR11 + %VAR10;
  //   %RET0 := %VAR11;

UserFunctionPou COORD_X
  (* SectionNumber=4, Description=%RET0: Coordenada en X
%PARAM0: Cuenta encoder L
%PARAM1: Cuenta encoder R *)

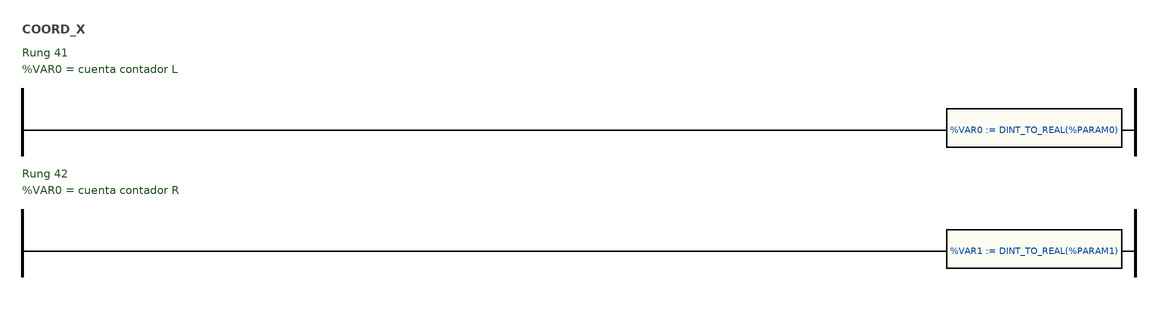

// Rung 41
// %VAR0 = cuenta contador L
  LD 1
  [%VAR0 := DINT_TO_REAL(%PARAM0)]
  // as ST:
  //   %VAR0 := DINT_TO_REAL(%PARAM0);

// Rung 42
// %VAR0 = cuenta contador R
  LD 1
  [%VAR1 := DINT_TO_REAL(%PARAM1)]
  // as ST:
  //   %VAR1 := DINT_TO_REAL(%PARAM1);

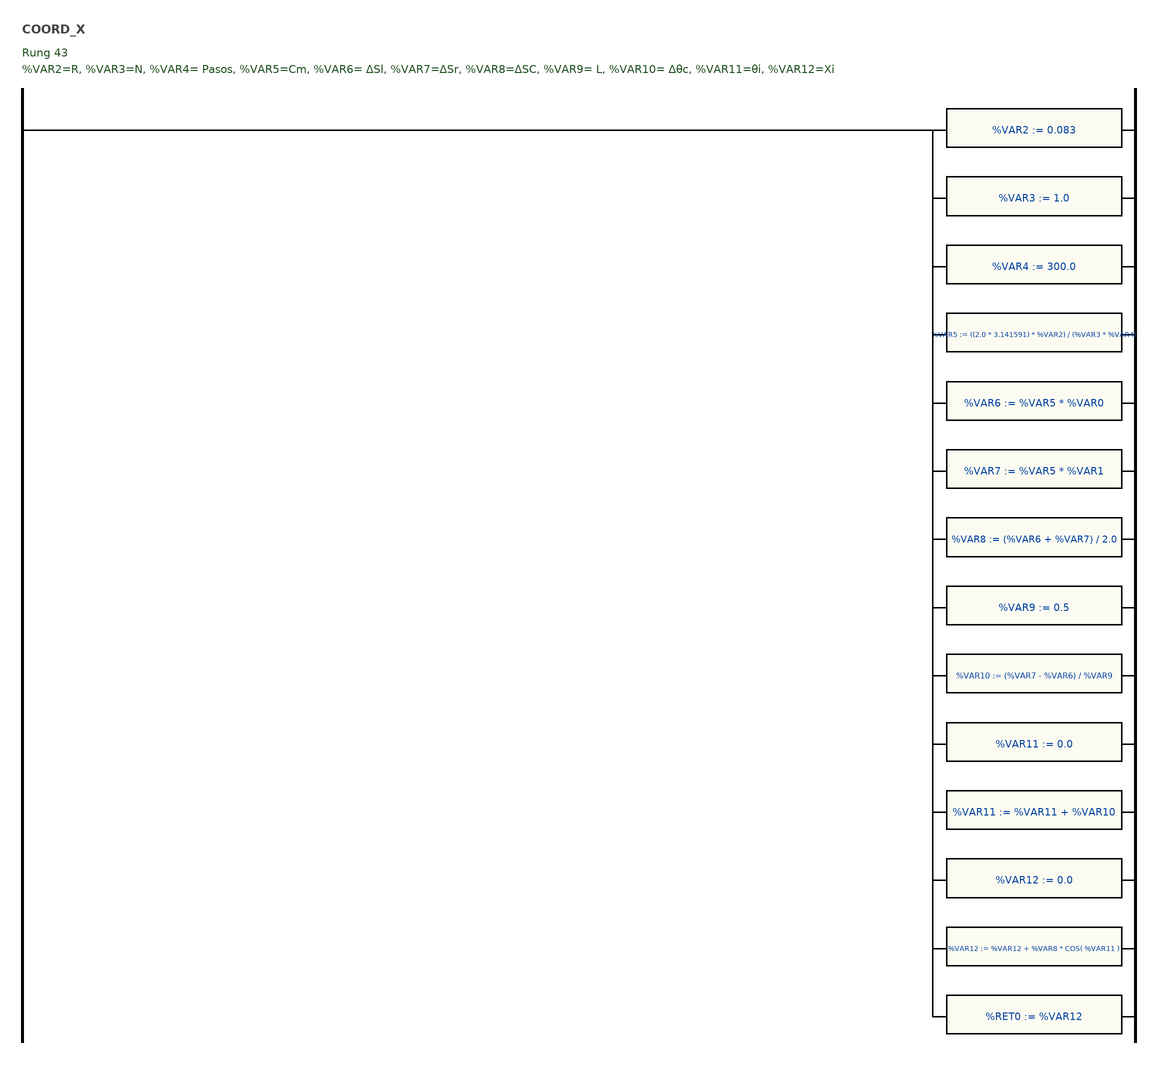

// Rung 43
// %VAR2=R, %VAR3=N, %VAR4= Pasos, %VAR5=Cm, %VAR6= ΔSl, %VAR7=ΔSr, %VAR8=ΔSC, %VAR9= L, %VAR10= Δθc, %VAR11=θi, %VAR12=Xi
  LD 1
  [%VAR2 := 0.083]
  [%VAR3 := 1.0]
  [%VAR4 := 300.0]
  [%VAR5 := ((2.0 * 3.141591) * %VAR2) / (%VAR3 * %VAR4)]
  [%VAR6 := %VAR5 * %VAR0]
  [%VAR7 := %VAR5 * %VAR1]
  [%VAR8 := (%VAR6 + %VAR7) / 2.0]
  [%VAR9 := 0.5]
  [%VAR10 := (%VAR7 - %VAR6) / %VAR9]
  [%VAR11 := 0.0]
  [%VAR11 := %VAR11 + %VAR10]
  [%VAR12 := 0.0]
  [%VAR12 := %VAR12 + %VAR8 * COS( %VAR11 )]
  [%RET0 := %VAR12]
  // as ST:
  //   %VAR2 := 0.083;
  //   %VAR3 := 1.0;
  //   %VAR4 := 300.0;
  //   %VAR5 := ((2.0 * 3.141591) * %VAR2) / (%VAR3 * %VAR4);
  //   %VAR6 := %VAR5 * %VAR0;
  //   %VAR7 := %VAR5 * %VAR1;
  //   %VAR8 := (%VAR6 + %VAR7) / 2.0;
  //   %VAR9 := 0.5;
  //   %VAR10 := (%VAR7 - %VAR6) / %VAR9;
  //   %VAR11 := 0.0;
  //   %VAR11 := %VAR11 + %VAR10;
  //   %VAR12 := 0.0;
  //   %VAR12 := %VAR12 + %VAR8 * COS( %VAR11 );
  //   %RET0 := %VAR12;

UserFunctionPou COORD_Y
  (* SectionNumber=3, Description=%RET0: Coordenada en Y
%PARAM0: Cuenta encoder L
%PARAM1: Cuenta encoder R *)

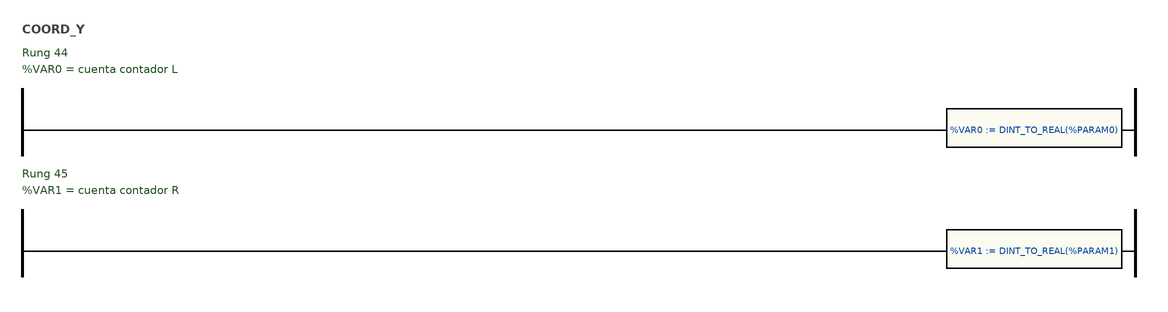

// Rung 44
// %VAR0 = cuenta contador L
  LD 1
  [%VAR0 := DINT_TO_REAL(%PARAM0)]
  // as ST:
  //   %VAR0 := DINT_TO_REAL(%PARAM0);

// Rung 45
// %VAR1 = cuenta contador R
  LD 1
  [%VAR1 := DINT_TO_REAL(%PARAM1)]
  // as ST:
  //   %VAR1 := DINT_TO_REAL(%PARAM1);

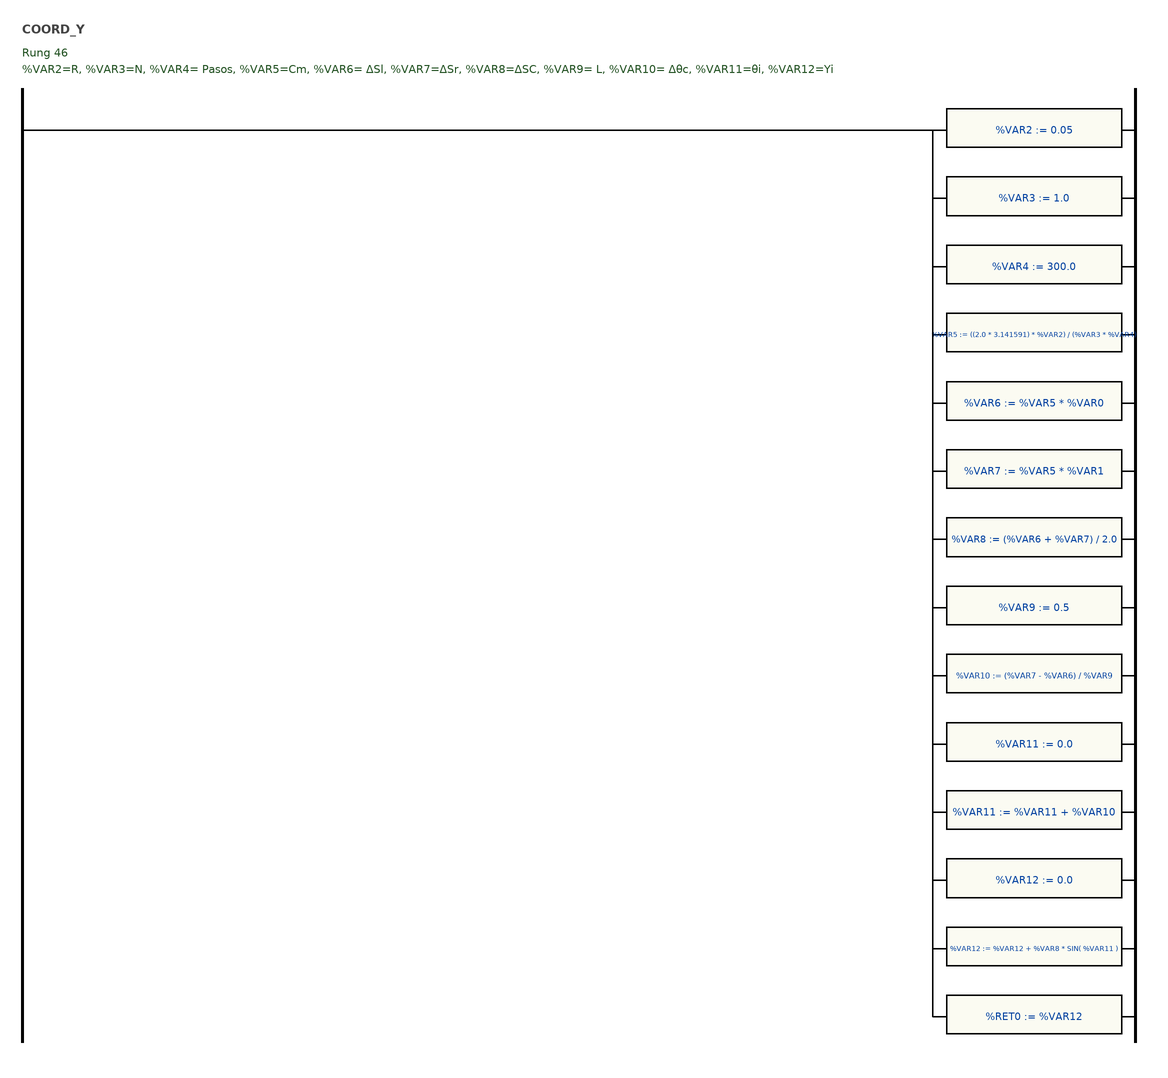

// Rung 46
// %VAR2=R, %VAR3=N, %VAR4= Pasos, %VAR5=Cm, %VAR6= ΔSl, %VAR7=ΔSr, %VAR8=ΔSC, %VAR9= L, %VAR10= Δθc, %VAR11=θi, %VAR12=Yi
  LD 1
  [%VAR2 := 0.05]
  [%VAR3 := 1.0]
  [%VAR4 := 300.0]
  [%VAR5 := ((2.0 * 3.141591) * %VAR2) / (%VAR3 * %VAR4)]
  [%VAR6 := %VAR5 * %VAR0]
  [%VAR7 := %VAR5 * %VAR1]
  [%VAR8 := (%VAR6 + %VAR7) / 2.0]
  [%VAR9 := 0.5]
  [%VAR10 := (%VAR7 - %VAR6) / %VAR9]
  [%VAR11 := 0.0]
  [%VAR11 := %VAR11 + %VAR10]
  [%VAR12 := 0.0]
  [%VAR12 := %VAR12 + %VAR8 * SIN( %VAR11 )]
  [%RET0 := %VAR12]
  // as ST:
  //   %VAR2 := 0.05;
  //   %VAR3 := 1.0;
  //   %VAR4 := 300.0;
  //   %VAR5 := ((2.0 * 3.141591) * %VAR2) / (%VAR3 * %VAR4);
  //   %VAR6 := %VAR5 * %VAR0;
  //   %VAR7 := %VAR5 * %VAR1;
  //   %VAR8 := (%VAR6 + %VAR7) / 2.0;
  //   %VAR9 := 0.5;
  //   %VAR10 := (%VAR7 - %VAR6) / %VAR9;
  //   %VAR11 := 0.0;
  //   %VAR11 := %VAR11 + %VAR10;
  //   %VAR12 := 0.0;
  //   %VAR12 := %VAR12 + %VAR8 * SIN( %VAR11 );
  //   %RET0 := %VAR12;
